// TIA Portal project "PLC1500" (V17)

(* hardware
DEVICE "S7-1500/ET200MP station_1"  S7-1500 station
   slot 0: "Rail_0"  Rack  6ES7 590-1***0-0AA0
   slot 1: "PLC_1"  CPU 1512C-1 PN  6ES7 512-1CK01-0AB0  V2.8
      slot 3: "CPU display_1"  6ES7591-1AA00-0AA0
      slot 32768: "PROFINET interface_1"  X1
         slot 32769: "Port_1"  X1 P1
         slot 32770: "Port_2"  X1 P2
      slot 34817: "Virtual CP interface port_1"  Virtual CP interface port  Virtual CP interface port
DEVICE "HMI_1"  TP700 Comfort
   slot 0: "HMI_1"  TP700 Comfort  6AV2 124-0GC01-0AX0  17.0.0.0
   slot 1: "HMI_RT_1"  TP700 Comfort  6AV2 124-0GC01-0AX0  17.0.0.0
   slot 5: "HMI_1.IE_CP_1"  PROFINET Interface  17.0.0.0
      slot 1: "PROFINET Interface_1"  PROFINET Interface
         slot 1: "Port_1"  Port
         slot 2: "Port_2"  Port
   slot 7: "HMI_1.MPI/DP_CP_1"  MPI/DP Interface  17.0.0.0
*)

// ===== PLC "PLC_1"  CPU 1512C-1 PN =====

VAR_GLOBAL   // PLC tag table "Default tag table"
   "Tag_1" AT %I10.0 : Bool;
   "Tag_2" AT %Q4.0 : Bool;
   "Tag_3" AT %I10.1 : Bool;
   "Tag_4" AT %Q4.1 : Bool;
   "Tag_5" AT %Q4.2 : Bool;
   "Tag_6" AT %M10.0 : Bool;
   "Tag_7" AT %M0.0 : Bool;
END_VAR

DATA_BLOCK "DB"   // DB2
{ S7_Optimized_Access := 'TRUE' }
VERSION : 0.1
   VAR
      disconnect : Bool;
      data : Array[0..10] of Int;
      connect : TCON_IP_v4;
   END_VAR
BEGIN
   connect.InterfaceId := 64;
   connect.ID := 1;
   connect.ConnectionType := 11;
   connect.LocalPort := 502;
END_DATA_BLOCK

DATA_BLOCK "DB_S7"   // DB3
{ S7_Optimized_Access := 'FALSE' }
VERSION : 0.1
   VAR
      thanhpho1 : String := '';
      thanhpho2 : String;
      thanhpho3 : String;
      setbit1 : Bool;
      Xylanh1 : Int;
      Xylanh2 : Int;
      Xylanh3 : Int;
   END_VAR
BEGIN
END_DATA_BLOCK

DATA_BLOCK "Chon_Tinh_ThanhPho_DB"   // DB4
{ S7_Optimized_Access := 'TRUE' }
VERSION : 0.1
// stored: InstanceOfName Chon_Tinh_ThanhPho
"Chon_Tinh_ThanhPho"
BEGIN
END_DATA_BLOCK

FUNCTION_BLOCK "Chon_Tinh_ThanhPho"   // FB1, LAD
{ S7_Optimized_Access := 'TRUE' }
VERSION : 0.1
BEGIN

REGION Network 1: Xylanh1
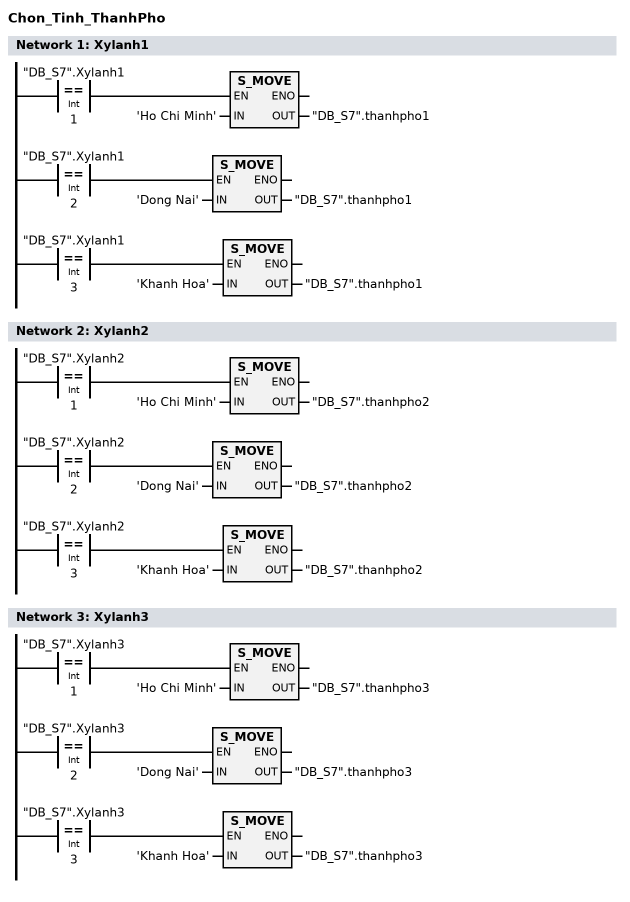
   RUNG wire#powerrail
      { S7_Templates := "SrcType := Int" } EQ_Contact(in1 := "DB_S7".Xylanh1, in2 := 1)
      S_Move(in := 'Ho Chi Minh', out => "DB_S7".thanhpho1)
   END_RUNG
   RUNG wire#powerrail
      { S7_Templates := "SrcType := Int" } EQ_Contact(in1 := "DB_S7".Xylanh1, in2 := 2)
      S_Move(in := 'Dong Nai', out => "DB_S7".thanhpho1)
   END_RUNG
   RUNG wire#powerrail
      { S7_Templates := "SrcType := Int" } EQ_Contact(in1 := "DB_S7".Xylanh1, in2 := 3)
      S_Move(in := 'Khanh Hoa', out => "DB_S7".thanhpho1)
   END_RUNG
   // the same network as SCL:
   IF "DB_S7".Xylanh1 = 1 THEN "DB_S7".thanhpho1 := 'Ho Chi Minh'; END_IF;
   IF "DB_S7".Xylanh1 = 2 THEN "DB_S7".thanhpho1 := 'Dong Nai'; END_IF;
   IF "DB_S7".Xylanh1 = 3 THEN "DB_S7".thanhpho1 := 'Khanh Hoa'; END_IF;
END_REGION

REGION Network 2: Xylanh2
   RUNG wire#powerrail
      { S7_Templates := "SrcType := Int" } EQ_Contact(in1 := "DB_S7".Xylanh2, in2 := 1)
      S_Move(in := 'Ho Chi Minh', out => "DB_S7".thanhpho2)
   END_RUNG
   RUNG wire#powerrail
      { S7_Templates := "SrcType := Int" } EQ_Contact(in1 := "DB_S7".Xylanh2, in2 := 2)
      S_Move(in := 'Dong Nai', out => "DB_S7".thanhpho2)
   END_RUNG
   RUNG wire#powerrail
      { S7_Templates := "SrcType := Int" } EQ_Contact(in1 := "DB_S7".Xylanh2, in2 := 3)
      S_Move(in := 'Khanh Hoa', out => "DB_S7".thanhpho2)
   END_RUNG
   // the same network as SCL:
   IF "DB_S7".Xylanh2 = 1 THEN "DB_S7".thanhpho2 := 'Ho Chi Minh'; END_IF;
   IF "DB_S7".Xylanh2 = 2 THEN "DB_S7".thanhpho2 := 'Dong Nai'; END_IF;
   IF "DB_S7".Xylanh2 = 3 THEN "DB_S7".thanhpho2 := 'Khanh Hoa'; END_IF;
END_REGION

REGION Network 3: Xylanh3
   RUNG wire#powerrail
      { S7_Templates := "SrcType := Int" } EQ_Contact(in1 := "DB_S7".Xylanh3, in2 := 1)
      S_Move(in := 'Ho Chi Minh', out => "DB_S7".thanhpho3)
   END_RUNG
   RUNG wire#powerrail
      { S7_Templates := "SrcType := Int" } EQ_Contact(in1 := "DB_S7".Xylanh3, in2 := 2)
      S_Move(in := 'Dong Nai', out => "DB_S7".thanhpho3)
   END_RUNG
   RUNG wire#powerrail
      { S7_Templates := "SrcType := Int" } EQ_Contact(in1 := "DB_S7".Xylanh3, in2 := 3)
      S_Move(in := 'Khanh Hoa', out => "DB_S7".thanhpho3)
   END_RUNG
   // the same network as SCL:
   IF "DB_S7".Xylanh3 = 1 THEN "DB_S7".thanhpho3 := 'Ho Chi Minh'; END_IF;
   IF "DB_S7".Xylanh3 = 2 THEN "DB_S7".thanhpho3 := 'Dong Nai'; END_IF;
   IF "DB_S7".Xylanh3 = 3 THEN "DB_S7".thanhpho3 := 'Khanh Hoa'; END_IF;
END_REGION
END_FUNCTION_BLOCK

ORGANIZATION_BLOCK "Main"   // OB1, LAD, ProgramCycle
TITLE = "Main Program Sweep (Cycle)"
{ S7_Optimized_Access := 'TRUE' }
VERSION : 0.1
   VAR_INPUT
      Initial_Call : Bool;   // Initial call of this OB
      Remanence : Bool;   // =True, if remanent data are available
   END_VAR
   VAR_TEMP   // added for the SCL form of the ladder/FBD networks
      _w1 : Bool;
   END_VAR
BEGIN

REGION Network 1
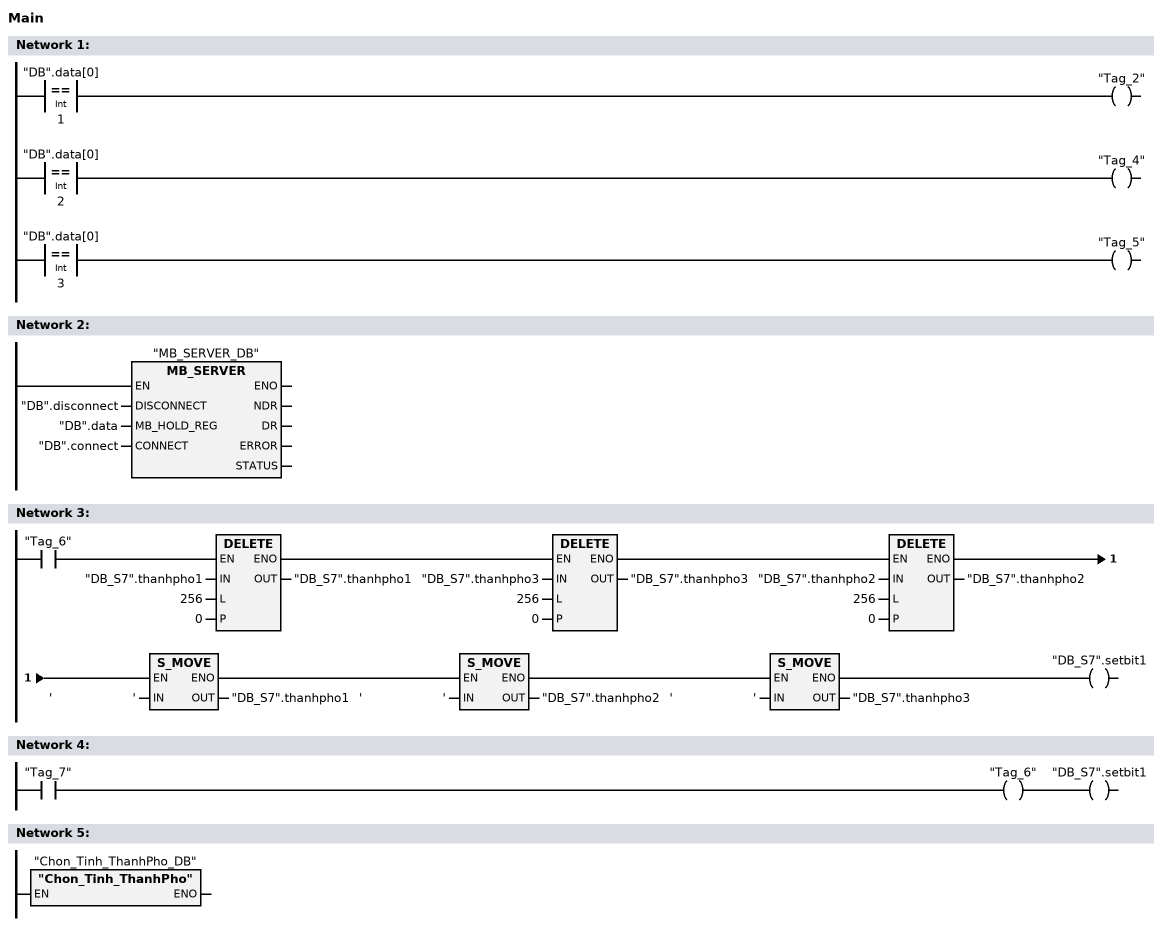
   RUNG wire#powerrail
      { S7_Templates := "SrcType := Int" } EQ_Contact(in1 := "DB".data[0], in2 := 1)
      Coil( "Tag_2" )
   END_RUNG
   RUNG wire#powerrail
      { S7_Templates := "SrcType := Int" } EQ_Contact(in1 := "DB".data[0], in2 := 2)
      Coil( "Tag_4" )
   END_RUNG
   RUNG wire#powerrail
      { S7_Templates := "SrcType := Int" } EQ_Contact(in1 := "DB".data[0], in2 := 3)
      Coil( "Tag_5" )
   END_RUNG
   // the same network as SCL:
   "Tag_2" := "DB".data[0] = 1;
   "Tag_4" := "DB".data[0] = 2;
   "Tag_5" := "DB".data[0] = 3;
END_REGION

REGION Network 2
   "MB_SERVER_DB"(DISCONNECT := "DB".disconnect, MB_HOLD_REG := "DB".data, CONNECT := "DB".connect);   // MB_SERVER
END_REGION

REGION Network 3
   #_w1 := "Tag_6";
   IF #_w1 THEN
       "DB_S7".thanhpho1 := DELETE(IN := "DB_S7".thanhpho1, L := 256, P := 0);
       "DB_S7".thanhpho3 := DELETE(IN := "DB_S7".thanhpho3, L := 256, P := 0);
       "DB_S7".thanhpho2 := DELETE(IN := "DB_S7".thanhpho2, L := 256, P := 0);
       "DB_S7".thanhpho1 := '                    ';
       "DB_S7".thanhpho2 := '                    ';
       "DB_S7".thanhpho3 := '                    ';
   END_IF;
   "DB_S7".setbit1 := #_w1;
END_REGION

REGION Network 4
   RUNG wire#powerrail
      Contact( "Tag_7" )
      Coil( "Tag_6" )
      Coil( "DB_S7".setbit1 )
   END_RUNG
   // the same network as SCL:
   "Tag_6" := "Tag_7";
   "DB_S7".setbit1 := "Tag_7";
END_REGION

REGION Network 5
   RUNG wire#powerrail
      "Chon_Tinh_ThanhPho_DB"()
   END_RUNG
   // the same network as SCL:
   "Chon_Tinh_ThanhPho_DB"();   // "Chon_Tinh_ThanhPho"
END_REGION
END_ORGANIZATION_BLOCK

(* ===== HMI "HMI_RT_1" =====
system functions are stored by id; their names below are inferred from use
connection "HMI_Connection_1": ETHERNET, S7_1500_OMS

HMI tags "Default tag table"
   "DB_S7_thanhpho1" : String[254] = PLC DB_S7.thanhpho1 AT %DB3.DBX0.0, 1 s
   "DB_S7_setbit1" : Bool = PLC DB_S7.setbit1 AT %DB3.DBX768.0, 1 s
   "DB_S7_Xylanh1" : Int = PLC DB_S7.Xylanh1 AT %DB3.DBW770, 1 s
   "DB_S7_Xylanh2" : Int = PLC DB_S7.Xylanh2 AT %DB3.DBW772, 1 s
   "DB_S7_Xylanh3" : Int = PLC DB_S7.Xylanh3 AT %DB3.DBW774, 1 s
   "Tag_7" : Bool = PLC Tag_7 AT %M0.0, 1 s
   "Tag_6" : Bool = PLC Tag_6 AT %M10.0, 1 s
   "Tag_2" : Bool = PLC Tag_2 AT %Q4.0, 1 s
   "Tag_4" : Bool = PLC Tag_4 AT %Q4.1, 1 s
   "Tag_5" : Bool = PLC Tag_5 AT %Q4.2, 1 s

text list "Text_list_1": 1 'Ho Chi Minh'; 2 'Dong Nai'; 3 'Khanh Hoa'

Template "Template_1" 800x480
   Button "Exit" at 720,420 size 78x58; TextOff 'Exit'; PictureOff "ExitRuntime_TP700_Comfort_TR"; PictureOn "ExitRuntime_TP700_Comfort_TR"
      on Release: StopRuntime(0)
   Button "Template_Button" at 640,420 size 78x58; TextOff 'Text'
   Button "Template_Button_1" at 560,420 size 78x58; TextOff 'Text'
   Button "Template_Button_2" at 480,420 size 78x58; TextOff 'Text'
   Button "Template_Button_3" at 400,420 size 78x58; TextOff 'Text'
   Button "Template_Button_4" at 321,420 size 78x58; TextOff 'Text'
   Button "Template_Button_5" at 241,420 size 78x58; TextOff 'Text'
   Button "Template_Button_6" at 161,420 size 78x58; TextOff 'Text'
   Button "Start screen" at 81,420 size 78x58; TextOff 'Start screen'; PictureOff "NavigateHome_TP700_Comfort_TR"; PictureOn "NavigateHome_TP700_Comfort_TR"
      on Release: ActivateScreen("Root screen", 0)
   Button "Alarms" at 1,420 size 78x58; TextOff 'Alarms'; PictureOff "AlarmDisplay_TP700_Comfort_TR"; PictureOn "AlarmDisplay_TP700_Comfort_TR"
      on Release: function_ef3f5d25("Alarm window_Unacknowledged", -1)

screen "Root screen" 800x480, template "Template_1"
   Button "Button_1" at 524,311 size 96x32; TextOff 'Reset'
      on Press: SetBit("Tag_6")
      on Release: ResetBit("Tag_6")
   Button "Button_2" at 220,311 size 96x32; TextOff 'Enter'
      on Press: SetBit("Tag_7")
      on Release: ResetBit("Tag_7")
   SymbolicIOField "Symbolic I/O field_1" at 62,144 size 170x32; TextOff '0'; TextOn '1'; TextList "Text_list_1"
      ProcessValue <- "DB_S7_Xylanh1"
   TextField "Text field_1" at 93,104 size 180x23; Text 'Xylanh 1'
   SymbolicIOField "Symbolic I/O field_2" at 329,144 size 170x32; TextOn '1'; TextOff '0'; TextList "Text_list_1"
      ProcessValue <- "DB_S7_Xylanh2"
   TextField "Text field_2" at 368,104 size 178x23; Text 'Xylanh 2'
   SymbolicIOField "Symbolic I/O field_3" at 595,144 size 170x32; TextOn '1'; TextOff '0'; TextList "Text_list_1"
      ProcessValue <- "DB_S7_Xylanh3"
   TextField "Text field_3" at 635,104 size 165x23; Text 'Xylanh 3'
   Circle "Circle_1" at 110,196 size 48x48
      Appearance <- "Tag_2"
   Circle "Circle_2" at 398,196 size 48x48
      Appearance <- "Tag_4"
   Circle "Circle_3" at 665,196 size 48x48
      Appearance <- "Tag_5"
   IOField "I/O field_1" at 177,28 size 96x32; FormatPattern ??????????
*)